ABB RAPID module: CalibData.modx

MODULE CalibData
    PERS tooldata Tool:=[TRUE,[[0,0,394],[1,0,0,0]],[1,[0,0,120],[1,0,0,0],0,0,0]];
    PERS wobjdata Workobject_1:=[FALSE,TRUE,"",[[247.143,3.713,1200],[0,1,0,0]],[[0,0,0],[1,0,0,0]]];
ENDMODULE
